(*			
	RAFALOS
	Rafał Osajda		19.09.2025		TC 4024.66
	
*)
FUNCTION_BLOCK FB_BaseLabel
VAR
	stTexts						: ST_Label;
END_VAR

METHOD PUBLIC GetText : WSTRING
VAR_INPUT
	eLocation				: E_Location;
END_VAR
GetText				:= THIS^.stTexts.arrText [eLocation];
END_METHOD

METHOD PUBLIC GetTexts : ST_Label
VAR_INPUT
END_VAR
GetTexts				:=THIS^.stTexts;
END_METHOD

METHOD PUBLIC SetText
VAR_INPUT
	eLocation			: E_Location;
	wsDescription		: WSTRING;
END_VAR
THIS^.stTexts.arrText [eLocation]	:= wsDescription;
END_METHOD

METHOD PUBLIC SetTexts
VAR_INPUT
	stTexts				: ST_Label;
END_VAR
THIS^.stTexts			:= stTexts;
END_METHOD

END_FUNCTION_BLOCK

(* stored: Version 1.1.0.1
   POU FB_BaseLabel: Id {e151c3ef-0d70-0a6d-3db5-a2f1d96fba32}, SpecialFunc None
   Method GetText: Id {a0c7ed25-2400-05ca-0002-fe2f26536c5f}
   Method GetTexts: Id {d80bba81-9353-01a2-25e9-143430746f38}
   Method SetText: Id {a325a82c-37c7-0885-1304-9e7776739f28}
   Method SetTexts: Id {ac0a0a67-d616-01b6-2ae1-e67d6995b8d6} *)
